{attribute 'GeneratedUsingTerminal: AT2050-0501-0019'}
{attribute addProperty BoxType "AT2050-0501-0019"}
{attribute addProperty Id "A_0081_AT2002_5250_0018_AT2002_5250AT2002_01D6DEDF80"}
{attribute addProperty CRC "2193275722"}
{attribute addProperty Size "80"}
TYPE A_0069_AT2050_0501_0019_AT2050_0501_82BABB4A EXTENDS AT2050_86175B41 :
STRUCT
	{attribute addProperty Name "A_0081_AT2002_5250_0018_AT2002_5250"}
	A_0081_AT2002_5250_0018_AT2002_5250 : AT2002_01D6DEDF;
END_STRUCT
END_TYPE

(* stored: Version 1.2.0.0, ProductVersion 3.1.4024.9
   DUT A_0069_AT2050_0501_0019_AT2050_0501_82BABB4A: Id {d87df239-10cb-43e1-a419-35ccbddf7abf} *)
